// TIA Portal V17 export
// export: Created 2025-08-05T09:35:56.4082252Z, ExportSetting WithDefaults, DisplayName Totally Integrated Automation Portal, DisplayVersion V17, DisplayName TIA Portal Openness, DisplayVersion V17, DisplayName TIA Portal Version Control Interface, DisplayVersion V17, DisplayName SINAMICS Startdrive Advanced, DisplayVersion V17, DisplayName SINAMICS Startdrive G130, G150, S120, S150, SINAMICS MV, S210, DisplayVersion V17, DisplayName SINAMICS Startdrive G110M, G120, G120C, G120D, G120P, G115D, DisplayVersion V17, DisplayName STEP 7 Professional, DisplayVersion V17, DisplayName STEP 7 Safety, DisplayVersion V17, DisplayName WinCC Advanced, DisplayVersion V17
FUNCTION_BLOCK "Call"   // FB1, LAD
{ S7_Optimized_Access := 'TRUE' }
VERSION : 0.1
// stored: AutoNumber true, IsIECCheckEnabled false, IsRetainMemResEnabled false, MemoryReserve 100, SetENOAutomatically false, UDAEnableTagReadback false
   VAR
      LaserComm_API_Instance { S7_SetPoint := 'True'} : Array[0..1] of "LaserComm_API";
      Dummy_Cereal_Number { S7_SetPoint := 'True'} : Array[1..32] of Char;
      Dummy_Part_Type { S7_SetPoint := 'True'} : Array[1..18] of Char;
   END_VAR
BEGIN

REGION Network 2: IPG and OPC FB Calls
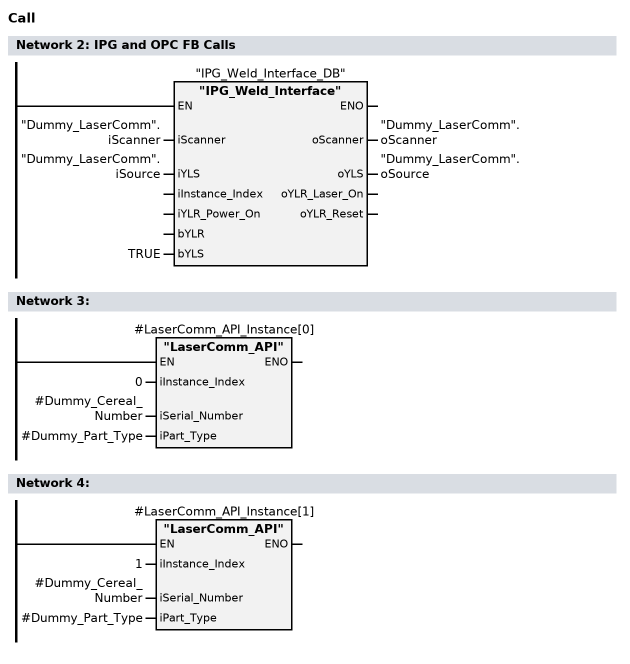
   RUNG wire#powerrail
      "IPG_Weld_Interface_DB"(iScanner := "Dummy_LaserComm".iScanner, iYLS := "Dummy_LaserComm".iSource, iInstance_Index :=, iYLR_Power_On :=, bYLR :=, bYLS := TRUE, oScanner => "Dummy_LaserComm".oScanner, oYLS => "Dummy_LaserComm".oSource, oYLR_Laser_On =>, oYLR_Reset =>)
   END_RUNG
   // the same network as SCL:
   "IPG_Weld_Interface_DB"(iScanner := "Dummy_LaserComm".iScanner,   // "IPG_Weld_Interface"
                           iYLS := "Dummy_LaserComm".iSource,
                           bYLS := TRUE,
                           oScanner => "Dummy_LaserComm".oScanner,
                           oYLS => "Dummy_LaserComm".oSource);
END_REGION

REGION Network 3
   RUNG wire#powerrail
      #LaserComm_API_Instance[0](iInstance_Index := 0, iSerial_Number := #Dummy_Cereal_Number, iPart_Type := #Dummy_Part_Type)
   END_RUNG
   // the same network as SCL:
   #LaserComm_API_Instance[0](iInstance_Index := 0,   // "LaserComm_API"
                           iSerial_Number := #Dummy_Cereal_Number,
                           iPart_Type := #Dummy_Part_Type);
END_REGION

REGION Network 4
   RUNG wire#powerrail
      #LaserComm_API_Instance[1](iInstance_Index := 1, iSerial_Number := #Dummy_Cereal_Number, iPart_Type := #Dummy_Part_Type)
   END_RUNG
   // the same network as SCL:
   #LaserComm_API_Instance[1](iInstance_Index := 1,   // "LaserComm_API"
                           iSerial_Number := #Dummy_Cereal_Number,
                           iPart_Type := #Dummy_Part_Type);
END_REGION
END_FUNCTION_BLOCK
